Universal Robots PolyScope program: program2.urp

Program program2 (installation=default directory=/ursim/programs createdIn=3.15.8.106339 lastSavedIn=3.15.8.106339 robotSerialNumber=2018359999)
Calibrated DH parameters: a=[0, -0.425, -0.39225, 0, 0, 0]; d=[0.089159, 0, 0, 0.10915, 0.09465, 0.0823]; alpha=[1.570796, 0, 0, 1.570796, -1.570796, 0]; deltaTheta=[0, 0, 0, 0, 0, 0]
Robot Program (runOnlyOnce=false)
  Script file /ursim/programs/programa2.script
    |   set_gravity([0.0, 0.0, 9.82])
    |   set_tcp(p[0.0,0.0,0.0,0.0,0.0,0.0])
    |   set_payload(2.0)
    |   set_tool_voltage(0)
    | 
    |   set_digital_out(0, True)
    | 
    |   popup("El control va a ser compartido con un controlador externo. Presione OK.", "Aviso", False, False, True)
    | 
    |   sleep(5.0)
    | 
    |   popup("Control compartido con ROS2. El robot está bajo control externo.", "Aviso", False, False, False)
    | 
    |   # Mantener el robot activo para recibir comandos externos
    |   while (True):
    |     sleep(0.1)
    |   end
